(* IEC 61131-3 sources: openplc-temperature-control/plc/temperature_control/pous/programs, 1 file *)

(* ---- main.st ---- *)
PROGRAM main
  VAR
    Temperature : UINT AT %MW0 := 20;
    Fan : BOOL AT %QX0.0 := FALSE;
  END_VAR

(* Cooling fan control with 3-degree hysteresis. *)

IF Temperature >= 30 THEN
    Fan := TRUE;
ELSIF Temperature <= 27 THEN
    Fan := FALSE;
END_IF;

END_PROGRAM
